// Mitsubishi GX Works2 project: plcdataword   PLC: Q03UDV

PROGRAM MAIN
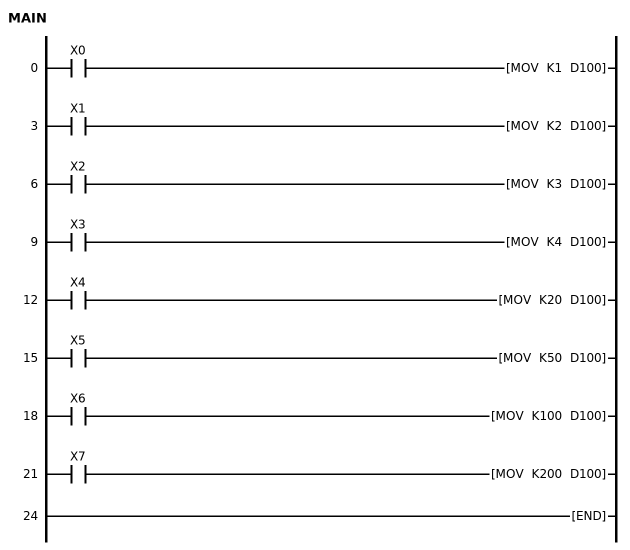
0     LD      X0
      MOV     K1 D100
3     LD      X1
      MOV     K2 D100
6     LD      X2
      MOV     K3 D100
9     LD      X3
      MOV     K4 D100
12    LD      X4
      MOV     K20 D100
15    LD      X5
      MOV     K50 D100
18    LD      X6
      MOV     K100 D100
21    LD      X7
      MOV     K200 D100
24    END
END_PROGRAM
